(* IEC 61131-3 sources: InfiniteStateMachine/extracted_st/project/infinitestatemachine/function_blocks, 1 file *)

(* ---- statemachine-StateMachine.st ---- *)
(* --- Interface --- *)
FUNCTION_BLOCK FINAL StateMachine
VAR_INPUT
END_VAR
VAR_OUTPUT
END_VAR
VAR
	itfStates : IStateArray;
	iDepth : INT := 0;
END_VAR
